{attribute 'linkalways'} 
{attribute 'no_explicit_call' := 'This FB is a CLASS and must be accessed using methods or properties'}
{attribute 'enable_dynamic_creation'}
FUNCTION_BLOCK Node_F_VN_SetPixels EXTENDS VisionNode
VAR
    ipDestImage : _ITcVnImage;
    aValue : _TcVnVector4_LREAL;
    hrPrev : _HRESULT(S_OK);
	hresult : _HRESULT(S_OK);
END_VAR

METHOD PUBLIC  Clone : I_Node
VAR
	pNode : POINTER TO Node_F_VN_SetPixels;
END_VAR
pNode := __NEW(Node_F_VN_SetPixels);
Clone := pNode^;
END_METHOD

METHOD FB_init : BOOL
VAR_INPUT
	bInitRetains : BOOL; // if TRUE, the retain variables are initialized (warm start / cold start)
	bInCopyCode : BOOL;  // if TRUE, the instance afterwards gets moved into the copy code (online change)
END_VAR
AddInput('ipDestImage', ipDestImage);
AddInput('aValue', aValue);
AddInput('hrPrev', hrPrev);
AddOutput('ipDestImage', ipDestImage);
AddOutput('hresult',hresult);
END_METHOD

METHOD PROTECTED  OnExecute : HRESULT
hresult.Value := F_VN_SetPixels(
    ipDestImage := ipDestImage.Value,
    aValue := aValue.Value,
	hrPrev:= hrPrev.Value);
END_METHOD

METHOD PUBLIC PreExecutionCheck
VAR_INPUT
	Check : I_PreExecutionChecks;
END_VAR
Check.IsTrue(ipDestImage.IsValid, 'ipDestImage must contain an image');
END_METHOD

END_FUNCTION_BLOCK

(* stored: Version 1.1.0.1, ProductVersion 3.1.4024.13
   POU Node_F_VN_SetPixels: Id {b3b16b4d-326a-09ff-3fc1-6f4433513a7f}, SpecialFunc None
   Folder Constructor: Id {894e75d9-764c-065a-1467-a99f9c46145f}
   Method Clone: Id {e07dde63-a505-02ea-0654-dcb44083212a}
   Method FB_init: Id {a34aab35-3bb9-0bcd-11c6-474a5ffde75c}
   Method OnExecute: Id {dd84eb0a-303b-0aa5-0e00-5013a6a1def6}
   Method PreExecutionCheck: Id {e24bef43-a85d-018f-3a3a-8c1dfdd073ae} *)
